Yaskawa INFORM job: R2_W08,11(-70,-90)_MP_OK.JBI

/JOB
//NAME R2_W08,11(-70,-90)_MP_OK
///FOLDERNAME MP_TEST
//POS
///NPOS 84,84,0,3,0,0
///TOOL 0
///POSTYPE PULSE
///PULSE
C00000=80634,56524,26439,-33552,116027,48375
C00001=80628,58269,45036,-31008,107028,51169
C00002=78911,55316,44053,-31183,105606,50866
C00003=78212,54208,43755,-31252,105015,50747
C00004=78077,53876,44572,-31170,104384,50872
C00005=78212,54208,43755,-31252,105015,50747
C00006=75675,58994,46299,-31860,104831,49753
C00007=75090,60550,48062,-31915,104366,49647
C00008=75675,58994,46299,-31860,104831,49753
C00009=73415,47128,27098,-33303,108822,47587
C00010=73012,45246,24655,-33476,109116,47321
C00011=73415,47128,27098,-33303,108822,47587
C00012=74150,48191,27319,-33287,109454,47700
C00013=75960,51015,28077,-33247,110987,47988
C00014=75965,52987,13601,-36257,119226,45094
C00015=136517,51935,5119,-1923,104393,8731
C00016=87157,-5483,-28306,57450,115604,41571
C00017=87147,-5039,-11335,53427,109619,37333
C00018=88649,-5898,-8462,52940,107396,36805
C00019=89258,-6153,-7236,52774,106498,36599
C00020=88843,-5700,-6906,52723,106753,36518
C00021=87960,-10028,-10339,52560,107187,36278
C00022=88843,-5700,-6906,52723,106753,36518
C00023=89258,-6153,-7236,52774,106498,36599
C00024=86366,24961,37253,63655,115225,35892
C00025=87245,23785,36110,63979,114710,36091
C00026=86366,24961,37253,63655,115225,35892
C00027=86261,20929,31425,64367,115990,36580
C00028=105942,-62521,-63510,26568,80862,38232
C00029=109708,-67430,-64024,26016,77688,38941
C00030=109885,-65154,-62228,25976,77691,39009
C00031=109708,-67430,-64024,26016,77688,38941
C00032=105942,-62521,-63510,26568,80862,38232
C00033=106960,-53147,-53640,26464,79409,38286
C00034=106853,-54251,-55854,26429,80158,38415
C00035=106579,-56879,-61286,26365,82039,38738
C00036=107641,-43424,-69167,26047,92329,41409
C00037=143143,24328,-21242,-15658,96224,-11878
C00038=72204,74256,59569,-26405,111997,60927
C00039=70917,68999,55676,-26710,111311,60566
C00040=85885,57876,53749,-32011,120623,64762
C00041=70563,68474,57156,-26581,110137,60710
C00042=70776,68944,56037,-26701,111041,60575
C00043=82327,65803,62898,-33102,117932,64007
C00044=66932,87982,79688,-30579,103155,62915
C00045=68273,94194,85253,-30231,103438,63379
C00046=67652,72456,53103,-19372,121960,51858
C00047=68730,81297,71878,-24437,120905,53913
C00048=70977,68393,57703,-23430,124019,52775
C00049=66315,67012,49556,-19800,121060,51456
C00050=65775,67263,51320,-19811,120027,51426
C00051=73586,65272,57175,-21672,123548,54069
C00052=68991,63069,47524,-18483,120952,52622
C00053=70206,68275,51151,-18045,121645,53017
C00054=67306,51124,50401,-20344,101560,40970
C00055=87477,30209,35148,-22218,113002,46164
C00056=84814,33924,44185,-23054,109360,46670
C00057=65224,53044,56715,-20613,98319,40767
C00058=65298,47795,50229,-20686,99552,40580
C00059=87649,41251,58483,-21198,105425,48508
C00060=71908,43018,52479,-24041,92531,45521
C00061=73734,43279,49847,-23760,94663,45760
C00062=75710,44802,35372,-24197,104128,44564
C00063=131785,47166,14001,-6017,108119,46057
C00064=158927,32103,13676,68669,79329,67442
C00065=158908,36411,34815,70732,75312,62704
C00066=161041,36978,37858,71079,73298,62259
C00067=161934,37353,39196,71241,72468,62082
C00068=161197,36103,37872,71200,73031,62071
C00069=161616,38399,39420,71134,72825,62225
C00070=160145,52009,60753,72851,71768,59260
C00071=159331,51665,59666,72650,72481,59393
C00072=157285,50529,55866,72065,74452,59955
C00073=158623,75600,58938,46322,103470,-39172
C00074=160646,74114,58732,46422,101973,-38891
C00075=161514,73751,58928,46458,101305,-38783
C00076=160874,72062,56896,46460,101906,-38810
C00077=161157,75917,61015,46390,101370,-38929
C00078=160543,87422,83058,45232,96249,-41626
C00079=159778,86810,81631,45169,97042,-41627
C00080=157799,88241,81814,44919,98490,-41911
C00081=156482,94558,73923,46181,104945,-39526
C00082=167679,39598,-22082,19335,97230,-42029
C00083=144689,40558,-40632,18601,81152,-34817
BC00000=15,149319,628321
BC00001=15,149319,628321
BC00002=15,149319,628321
BC00003=15,149319,628321
BC00004=15,149319,628321
BC00005=15,149319,628321
BC00006=15,149319,628321
BC00007=15,149319,628321
BC00008=15,149319,628321
BC00009=15,149319,628321
BC00010=15,149319,628321
BC00011=15,149319,628321
BC00012=15,149319,628321
BC00013=15,149319,628321
BC00014=15,149319,628321
BC00015=161990,237162,590954
BC00016=74827,184870,688957
BC00017=74827,184870,688957
BC00018=74827,184870,688957
BC00019=74827,184870,688957
BC00020=74827,184870,688957
BC00021=74827,184870,688957
BC00022=74827,184870,688957
BC00023=74827,184870,688957
BC00024=74827,184870,688957
BC00025=74827,184870,688957
BC00026=74827,184870,688957
BC00027=74827,184870,688957
BC00028=74827,184870,688957
BC00029=74827,184870,688957
BC00030=74827,184870,688957
BC00031=74827,184870,688957
BC00032=74827,184870,688957
BC00033=74827,184870,688957
BC00034=74827,184870,688957
BC00035=74827,184870,688957
BC00036=74827,184870,688957
BC00037=161990,226164,590954
BC00038=18200,151858,666099
BC00039=18200,151858,666099
BC00040=64204,151857,666090
BC00041=18200,151858,666099
BC00042=18200,151858,666099
BC00043=77068,151857,666090
BC00044=18200,151858,666099
BC00045=18200,151858,666099
BC00046=26785,141685,638446
BC00047=26785,141685,638446
BC00048=39931,141685,638446
BC00049=26785,141685,638446
BC00050=26785,141685,638446
BC00051=39931,141685,638446
BC00052=26785,141685,638446
BC00053=26785,141685,638446
BC00054=7685,134768,792502
BC00055=68177,134768,792502
BC00056=64162,134768,792502
BC00057=7685,134768,792502
BC00058=7685,134768,792502
BC00059=64162,134768,792502
BC00060=7685,134768,792502
BC00061=7685,134768,792502
BC00062=7685,134768,792502
BC00063=125249,229988,669995
BC00064=278947,187063,652650
BC00065=278947,187063,652650
BC00066=278947,187063,652650
BC00067=278947,187063,652650
BC00068=278947,187063,652650
BC00069=278947,187063,652650
BC00070=278947,187063,652650
BC00071=278947,187063,652650
BC00072=278947,187063,652650
BC00073=259918,180997,570644
BC00074=259918,180997,570644
BC00075=259918,180997,570644
BC00076=259918,180997,570644
BC00077=259918,180997,570644
BC00078=259918,180997,570644
BC00079=259918,180997,570644
BC00080=259918,180997,570644
BC00081=259918,180997,570644
BC00082=259919,180998,570641
BC00083=239349,329429,575206
///POSTYPE BASE
///RECTAN
///RCONF 0,0,0,0,0,0,0,0,0,0,0,0,0,0,0,0,0,0,0,0,0,0,0,0
P00006=0.222,-3.123,-1.508,0.0000,0.0000,0.0000
P00021=-0.225,-6.128,-0.405,0.0000,0.0000,0.0000
P00026=0.562,-0.002,-0.337,0.0000,0.0000,0.0000
//INST
///DATE 2023/11/16 13:51
///ATTR SC,RW
///GROUP1 RB1,BS1
NOP
'r2_W08,11(-70,-90)
'Path S787 (for W8)
SFTOF
MOVJ C00000 BC00000 VJ=20.00
MOVJ C00001 BC00001 VJ=20.00
MOVL C00002 BC00002 V=100.0
MOVL C00003 BC00003 V=60.0
REFP 3 C00004 BC00004
CALL JOB:SEARCH-R1
SET P021 P006
SFTON P021
MOVL C00005 BC00005 V=60.0
MOVL C00006 BC00006 V=60.0
REFP 3 C00007 BC00007
CALL JOB:SEARCH-R1
SET P021 P006
SFTON P021
MOVL C00008 BC00008 V=60.0
MOVL C00009 BC00009 V=60.0
REFP 3 C00010 BC00010
CALL JOB:SEARCH-R1
SET P021 P006
SFTON P021
MOVL C00011 BC00011 V=60.0
MOVL C00012 BC00012 V=100.0
MOVL C00013 BC00013 V=100.0
MOVL C00014 BC00014 V=100.0
MOVJ C00015 BC00015 VJ=20.00
'Path S867
SFTOF
MOVJ C00016 BC00016 VJ=20.00
MOVJ C00017 BC00017 VJ=20.00
MOVL C00018 BC00018 V=100.0
MOVL C00019 BC00019 V=100.0
MOVL C00020 BC00020 V=60.0
REFP 3 C00021 BC00021
CALL JOB:SEARCH-R1
SET P026 P006
SFTON P026
MOVL C00022 BC00022 V=60.0
MOVL C00023 BC00023 V=100.0
MOVL C00024 BC00024 V=60.0
REFP 3 C00025 BC00025
CALL JOB:SEARCH-R1
SET P026 P006
SFTON P026
MOVL C00026 BC00026 V=60.0
MOVL C00027 BC00027 V=100.0
MOVL C00028 BC00028 V=100.0
MOVL C00029 BC00029 V=60.0
REFP 3 C00030 BC00030
CALL JOB:SEARCH-R1
SET P026 P006
SFTON P026
MOVL C00031 BC00031 V=60.0
MOVL C00032 BC00032 V=100.0
MOVL C00033 BC00033 V=100.0
MOVL C00034 BC00034 V=100.0
MOVL C00035 BC00035 V=100.0
MOVL C00036 BC00036 V=100.0
MOVJ C00037 BC00037 VJ=20.00
'Path W5
SFTOF
SFTON P021
MOVJ C00038 BC00038 VJ=20.00
MOVL C00039 BC00039 V=100.0
MOVL C00040 BC00040 V=100.0 PL=0
REFP 1 C00041 BC00041
REFP 2 C00042 BC00042
MACRO1 MJ#(0) ARGF6
ARCON
MOVL C00043 BC00043 V=8.3
ARCOF
MOVL C00044 BC00044 V=100.0
MOVL C00045 BC00045 V=100.0
SFTOF
'Path W6
SFTOF
SFTON P021
MOVJ C00046 BC00046 VJ=20.00
MOVL C00047 BC00047 V=100.0
MOVL C00048 BC00048 V=100.0 PL=0
REFP 1 C00049 BC00049
REFP 2 C00050 BC00050
MACRO1 MJ#(0) ARGF6
ARCON
MOVL C00051 BC00051 V=8.3
ARCOF
MOVL C00052 BC00052 V=100.0
MOVL C00053 BC00053 V=100.0
SFTOF
'Path W7
SFTOF
SFTON P021
MOVJ C00054 BC00054 VJ=20.00
MOVL C00055 BC00055 V=100.0
MOVL C00056 BC00056 V=100.0 PL=0
REFP 1 C00057 BC00057
REFP 2 C00058 BC00058
MACRO1 MJ#(0) ARGF6
ARCON
MOVL C00059 BC00059 V=8.3
ARCOF
MOVL C00060 BC00060 V=100.0
MOVL C00061 BC00061 V=100.0
MOVL C00062 BC00062 V=100.0
SFTOF
MOVJ C00063 BC00063 VJ=20.00
'
'Path W8
SFTOF
SFTON P026
MOVJ C00064 BC00064 VJ=20.00
MOVJ C00065 BC00065 VJ=20.00
MOVL C00066 BC00066 V=100.0
MOVL C00067 BC00067 V=100.0 PL=0
REFP 1 C00068 BC00068
REFP 2 C00069 BC00069
MACRO1 MJ#(0) ARGF6
ARCON
MOVL C00070 BC00070 V=8.3
ARCOF
MOVL C00071 BC00071 V=100.0
MOVL C00072 BC00072 V=100.0
SFTOF
'Path W868
SFTOF
SFTON P026
MOVJ C00073 BC00073 VJ=20.00
MOVL C00074 BC00074 V=100.0
MOVL C00075 BC00075 V=100.0 PL=0
REFP 1 C00076 BC00076
REFP 2 C00077 BC00077
MACRO1 MJ#(0) ARGF6
ARCON
MOVL C00078 BC00078 V=8.3
ARCOF
MOVL C00079 BC00079 V=100.0
MOVL C00080 BC00080 V=100.0
MOVL C00081 BC00081 V=100.0
SFTOF
MOVJ C00082 BC00082 VJ=20.00
MOVJ C00083 BC00083 VJ=20.00
END
